VAR_GLOBAL
	Scope_TempCtrlVariables					: FB_Scope_TempCtrlVariables;
END_VAR

(* stored: Version 1.1.0.1, ProductVersion 3.1.4024.12
   GVL GVL_30_Scope: Id {eae30708-51e6-42d1-a1c7-5b5eea3db711} *)
